TYPE "Pump"
VERSION : 0.1
   STRUCT
      Q : Bool;
      IsRunning : Bool;
      HasError : Bool;
   END_STRUCT;

END_TYPE

